(* PLC project CoDeSys External Library Template, WAGO e!COCKPIT e!COCKPIT, author 3S - Smart Software Solutions GmbH *)
(* stored: creationDateTime 2019-10-29T12:22:40.4862616, version 3.5.5.30, modificationDateTime 2019-10-24T14:40:07.960949, organization 3S - Smart Software Solutions GmbH *)
(* Library project template with all possible element types, docu and a sample project structure *)

(* values of enumPPPSWezelClimatixPOL63xErrorKlasa: AlarmCzujnikaZewnetrznego: alarm braku zmiany wartości czujnika temp. zewnetrznj; AlarmCzujnikaZasilaniaObwoduHC1: alarm braku zmiany wartości czujnika temp. zasilana obwodu HC1; AlarmCzujnikaZasilaniaObwoduDHW: alarm braku zmiany wartości czujnika temp. zasilana obwodu DHW; AlarmBrakuOsiagnieciaTemperaturyHC1: alarm braku osiągnięcia temp. zadanej obwodu HC1; AlarmBrakuOsiagnieciaTemperaturyDHW: alarm braku osiągnięcia temp. zadanej obwodu DHW; BladIloscPomiarowTemperatury: alarm zbyt małej ilości pomiarów dokonanych w ciągu dnia do obliczenia średniej *)

(* Autor: Paweł Kąkol, 2018-09-03-PK Prawa majątkowe: Solwena Sp. z o.o., Aktualizacje: 2019-02-14-AWy: dodanie alarmów czujników temp. zewnętrznej i zasilania obwodu HC1, DHW 2019-02-18-AWy: zmiana klas alarmów Opis: enum służy do definicji klas alarmów w fb węzła Climatix POL63x na budynkach PPP Sopot (ENGIE) *)
{attribute 'qualified_only'}
{attribute 'strict'}
TYPE enumPPPSWezelClimatixPOL63xErrorKlasa : (BrakKomunikacji := enumKlasaAlarmu.AwariaAutomatyki, AlarmOgolnyBezpieczenstwa := enumKlasaAlarmu.Bezpieczenstwa, AlarmOgolnyKrytyczny := enumKlasaAlarmu.Krytyczny, AlarmOgolnyOstrzezenie := enumKlasaAlarmu.Ostrzezenie, AlarmOgolnyInformacyjny := enumKlasaAlarmu.Informacyjny, AlarmCzujnikaZewnetrznego := enumKlasaAlarmu.AwariaAutomatyki, AlarmCzujnikaZasilaniaObwoduHC1 := enumKlasaAlarmu.AwariaAutomatyki, AlarmCzujnikaZasilaniaObwoduDHW := enumKlasaAlarmu.AwariaAutomatyki, AlarmBrakuOsiagnieciaTemperaturyHC1 := enumKlasaAlarmu.Ostrzezenie, AlarmBrakuOsiagnieciaTemperaturyDHW := enumKlasaAlarmu.Ostrzezenie, BladIloscPomiarowTemperatury := enumKlasaAlarmu.AwariaAutomatyki);
END_TYPE
